{attribute 'OPC.UA.DA.JobMethod' := 'JobMethode_CompressorControl'}
FUNCTION_BLOCK VSG_AS_CompressorControl
VAR
	AlwaysTrue : BOOL := TRUE;
	// Used for debugging purposes to display InputArguments of method call
	MethodCall_CompressorControl : BOOL := FALSE; // used to store InputArg "MethodCall" from Start() method
	Destination : BOOL;
	EncoderTargetPosition_01 : BOOL;
	EncoderTargetPosition_02 : BOOL;
	EncoderTargetPosition_03 : BOOL;
	EncoderTargetPosition_04 : BOOL;
	EncoderTargetPosition_05 : BOOL;
	EncoderTargetPosition_06 : BOOL;
	TS_EndschalterEntlastung : BOOL;
	callCounterStart : ULINT; // counts how many times the Start() method has been called
	callCounterCheckState : ULINT; // counts how many times the CheckState() method has been called
	callCounterAbort : ULINT; // counts how many times the Abort() method has been called
	
	// Variables to determine if a job has been started (Start() method has been called) or finished
	jobRunning : BOOL;
	jobFinished : BOOL;

	// State machine variable
	state : UDINT;
	
	//Variablen des Transport FBs
	ResetCall : BOOL := FALSE;	
	MBS_VSG_VerticalMove : CompressorControl;
END_VAR
	
VAR_INPUT
	NotAusSignal: BOOL;
//	LightSensor_01 : BOOL;
//	LightSensor_02 : BOOL;
//	TS_Endschalter_01 : BOOL;
//	TS_Endschalter_02 : BOOL;
	EncoderStartPosition_01 : BOOL;
	EncoderStartPosition_02 : BOOL;
	EncoderStartPosition_03 : BOOL;
	EncoderStartPosition_04 : BOOL;
	EncoderStartPosition_05 : BOOL;
	EncoderStartPosition_06 : BOOL;
	PowerOnDelay_Compressor : TIME;
	PowerOnDelay_Ventil : TIME;
END_VAR

VAR_OUTPUT
	Compressor : BOOL;
	Ventil : BOOL;
END_VAR

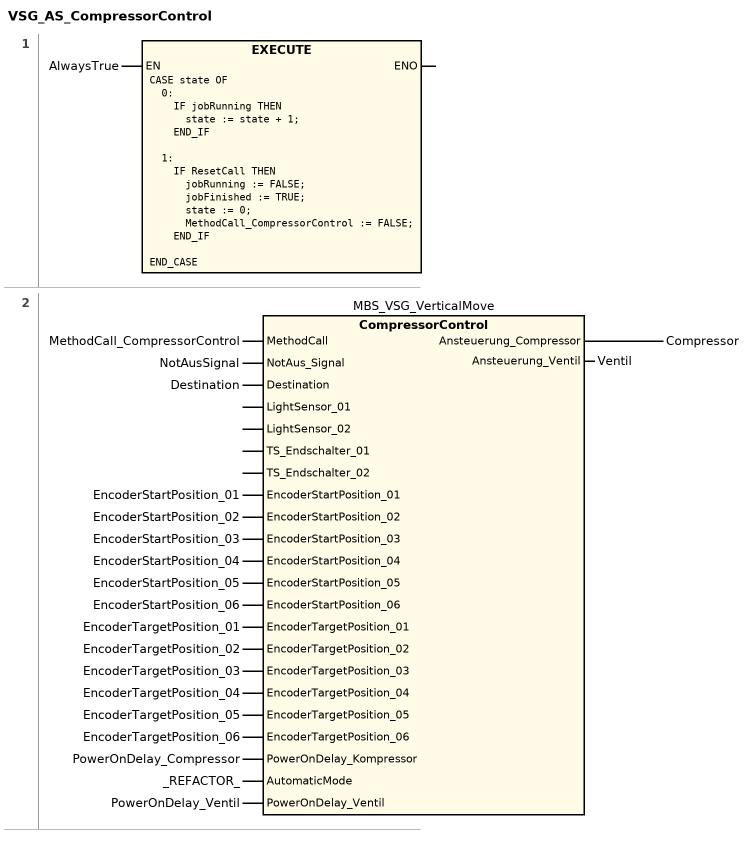
// NETWORK 1
IF AlwaysTrue THEN
    CASE state OF
    	0:
    		IF jobRunning THEN
    			state := state + 1;
    		END_IF
    		
    	1:
    		IF ResetCall THEN
    			jobRunning := FALSE;
    			jobFinished := TRUE;
    			state := 0;
    			MethodCall_CompressorControl := FALSE;
    		END_IF
    		
    END_CASE
END_IF

// NETWORK 2
MBS_VSG_VerticalMove(
    MethodCall := MethodCall_CompressorControl,
    NotAus_Signal := NotAusSignal,
    Destination := Destination,
    EncoderStartPosition_01 := EncoderStartPosition_01,
    EncoderStartPosition_02 := EncoderStartPosition_02,
    EncoderStartPosition_03 := EncoderStartPosition_03,
    EncoderStartPosition_04 := EncoderStartPosition_04,
    EncoderStartPosition_05 := EncoderStartPosition_05,
    EncoderStartPosition_06 := EncoderStartPosition_06,
    EncoderTargetPosition_01 := EncoderTargetPosition_01,
    EncoderTargetPosition_02 := EncoderTargetPosition_02,
    EncoderTargetPosition_03 := EncoderTargetPosition_03,
    EncoderTargetPosition_04 := EncoderTargetPosition_04,
    EncoderTargetPosition_05 := EncoderTargetPosition_05,
    EncoderTargetPosition_06 := EncoderTargetPosition_06,
    PowerOnDelay_Kompressor := PowerOnDelay_Compressor,
    AutomaticMode := _REFACTOR_,
    PowerOnDelay_Ventil := PowerOnDelay_Ventil,
    Ansteuerung_Ventil => Ventil); // CompressorControl
Compressor := MBS_VSG_VerticalMove.Ansteuerung_Compressor;

{attribute 'TcRpcEnable' := '1'}
METHOD Abort : HRESULT
VAR_INPUT
	hdl : UDINT; // Do not change, used by server.
END_VAR
callCounterAbort := callCounterAbort + 1;
END_METHOD

{attribute 'TcRpcEnable' := '1'}
METHOD CheckState : HRESULT
VAR_INPUT
	hdl : UDINT; // Do not change, used by server.
END_VAR
VAR_OUTPUT
	bBusy : BOOL; // Do not change. Used by server to find out if the job is finished
	
	// List of OutputArguments for OPC UA method, may be customized
	State : BOOL; // Abgeschlossener MethodCall
	MethodCall: BOOL; //Input Recall
END_VAR
callCounterCheckState := callCounterCheckState + 1;
IF NOT jobFinished THEN
	bBusy := TRUE; // job is not finished yet
	CheckState := 0; // no error
ELSE
	bBusy := FALSE; // job is finished
	CheckState := 0; // done, no error occured during execution (OPC UA StatusCode "GOOD")
	jobFinished := FALSE;
	State := ResetCall;
	MethodCall := MethodCall_CompressorControl;
END_IF
END_METHOD

{attribute 'TcRpcEnable' := '1'}
METHOD Start : HRESULT
VAR_INPUT
	// List of InputArguments for OPC UA method, may be customized
	MethodCall : BOOL; // some description
	Destination : BOOL;
	EncoderValueHorizontal_01 : BOOL;
	EncoderValueHorizontal_02 : BOOL;
	EncoderValuetVertical_01 : BOOL;
	EncoderValuetVertical_02 : BOOL;
	EncoderValuetRotation_01 : BOOL;	
	EncoderValuetRotation_02 : BOOL;
END_VAR
VAR_OUTPUT
	hdl : UDINT; // Do not change, used by server.
END_VAR
callCounterStart := callCounterStart + 1;

MethodCall_CompressorControl := MethodCall;
Destination := Destination;
//Ecoder Target Position Values
EncoderTargetPosition_01 := EncoderValueHorizontal_01;
EncoderTargetPosition_02 := EncoderValueHorizontal_02;
EncoderTargetPosition_03 := EncoderValuetVertical_01;
EncoderTargetPosition_04 := EncoderValuetVertical_02;
EncoderTargetPosition_05 := EncoderValuetRotation_01;
EncoderTargetPosition_06 := EncoderValuetRotation_02;

jobRunning := TRUE;
Start := 0; // no error occured, e.g. while parsing the input arguments (0 = OPC UA StatusCode "GOOD")
END_METHOD

END_FUNCTION_BLOCK

(* stored: Version 1.1.0.1, ProductVersion 3.1.4024.15
   POU VSG_AS_CompressorControl: Id {4cc652b0-658e-4a3b-ab9d-9b5203bcf388}, SpecialFunc None
   Method Abort: Id {5e67d4be-a065-4326-8feb-f9c7c95d4fa3}
   Method CheckState: Id {aefd6509-8302-4cce-ab29-0cbec4ce8596}
   Method Start: Id {75b53eb3-7bcb-463f-a353-7daeba059626} *)
